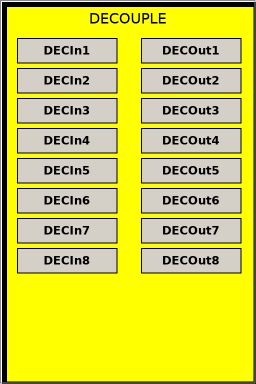
VISUALIZATION V_PH_DECOUPLE  // 256x384
VAR_INPUT
	stSafetyDecouple			: ST_SAFETY_FBDECOUPLE;
END_VAR
    Rectangle (2,2 256x384), colour toggle: stSafetyDecouple.bGeneralError
    Label (5,6 246x25), "DECOUPLE"
    RoundedRectangle (17,38 100x25), "DECIn1", colour toggle: stSafetyDecouple.uStatus.stStatusWords.wInputs.8
    RoundedRectangle (17,98 100x25), "DECIn3", colour toggle: stSafetyDecouple.uStatus.stStatusWords.wInputs.10
    RoundedRectangle (17,158 100x25), "DECIn5", colour toggle: stSafetyDecouple.uStatus.stStatusWords.wInputs.12
    RoundedRectangle (17,218 100x25), "DECIn7", colour toggle: stSafetyDecouple.uStatus.stStatusWords.wInputs.14
    RoundedRectangle (17,188 100x25), "DECIn6", colour toggle: stSafetyDecouple.uStatus.stStatusWords.wInputs.13
    RoundedRectangle (17,68 100x25), "DECIn2", colour toggle: stSafetyDecouple.uStatus.stStatusWords.wInputs.9
    RoundedRectangle (17,128 100x25), "DECIn4", colour toggle: stSafetyDecouple.uStatus.stStatusWords.wInputs.11
    RoundedRectangle (17,248 100x25), "DECIn8", colour toggle: stSafetyDecouple.uStatus.stStatusWords.wInputs.15
    RoundedRectangle (141,38 100x25), "DECOut1", colour toggle: stSafetyDecouple.uStatus.stStatusWords.wOutputs.8
    RoundedRectangle (141,68 100x25), "DECOut2", colour toggle: stSafetyDecouple.uStatus.stStatusWords.wOutputs.9
    RoundedRectangle (141,98 100x25), "DECOut3", colour toggle: stSafetyDecouple.uStatus.stStatusWords.wOutputs.10
    RoundedRectangle (141,128 100x25), "DECOut4", colour toggle: stSafetyDecouple.uStatus.stStatusWords.wOutputs.11
    RoundedRectangle (141,188 100x25), "DECOut6", colour toggle: stSafetyDecouple.uStatus.stStatusWords.wOutputs.13
    RoundedRectangle (141,158 100x25), "DECOut5", colour toggle: stSafetyDecouple.uStatus.stStatusWords.wOutputs.12
    RoundedRectangle (141,218 100x25), "DECOut7", colour toggle: stSafetyDecouple.uStatus.stStatusWords.wOutputs.14
    RoundedRectangle (141,248 100x25), "DECOut8", colour toggle: stSafetyDecouple.uStatus.stStatusWords.wOutputs.15
    Textfield (17,354 234x25), text list: 'TL_FbState', text index: stSafetyDecouple.eState
END_VISUALIZATION

(* stored: Version 1.1.0.1, ProductVersion 3.1.4024.4
   Visu V_PH_DECOUPLE: Id {c081c4f4-cc71-41b8-8d99-10fc24ddfd4a} *)
